Yaskawa INFORM job: FRONT_OST.JBI

/JOB
//NAME FRONT_OST
//POS
///NPOS 25,25,0,5,0,0
///TOOL 0
///POSTYPE PULSE
///PULSE
C00000=27585,-47842,-289,32095,-40789,28095
C00001=4801,-35772,25187,4593,-28023,-82032
C00002=17634,-23800,39238,9573,-31425,-73339
C00003=17634,-23800,39238,9573,-31425,-73339
C00004=16549,-22464,39800,8390,-30730,-72975
C00005=16684,-22641,39722,8536,-30818,-73021
C00006=16684,-19968,45512,8078,-32771,-72767
C00007=17634,-23800,39238,9573,-31425,-73339
C00008=17837,-21535,44509,9322,-33342,-73155
C00009=17837,-21535,44509,9322,-33342,-73155
C00010=16866,-20378,45014,8305,-32755,-72853
C00011=17032,-20588,44918,8481,-32857,-72905
C00012=17032,-17542,51480,8009,-35060,-72636
C00013=17837,-21535,44509,9322,-33342,-73155
C00014=-20829,-18800,50532,-12466,-37179,-77446
C00015=-19934,-17904,50946,-11618,-36715,-77676
C00016=-20044,-18019,50891,-11723,-36773,-77647
C00017=-20044,-15288,56753,-11218,-38713,-77950
C00018=-20966,-18928,50473,-12596,-37250,-77413
C00019=-20884,-26676,33664,-14451,-31668,-76336
C00020=-20884,-26676,33664,-14451,-31668,-76336
C00021=-19557,-25338,34176,-13080,-30873,-76751
C00022=-19691,-25483,34117,-13220,-30955,-76709
C00023=-19691,-22773,39998,-12506,-32911,-77106
C00024=-20642,-26447,33747,-14206,-31526,-76411
BC00000=934475
BC00001=880430
BC00002=895791
BC00003=895791
BC00004=895791
BC00005=895791
BC00006=895791
BC00007=895791
BC00008=900237
BC00009=900237
BC00010=900237
BC00011=900237
BC00012=900237
BC00013=900237
BC00014=900237
BC00015=900237
BC00016=900237
BC00017=900237
BC00018=900237
BC00019=900237
BC00020=900237
BC00021=900237
BC00022=900237
BC00023=900237
BC00024=900237
///POSTYPE BASE
///RECTAN
///RCONF 1,0,0,0,0,0,0,0,0,0,0,0,0,0,0,0,0,0,0,0,0,0,0,0
P00006=0.000,0.000,0.000,0.0000,0.0000,0.0000
///RCONF 0,0,0,0,0,0,0,0,0,0,0,0,0,0,0,0,0,0,0,0,0,0,0,0
P00021=6.550,-0.003,-5.735,0.0000,0.0000,0.0000
P00022=5.943,-0.018,-6.388,0.0000,0.0000,0.0000
P00023=7.025,-0.019,-7.168,0.0000,0.0000,0.0000
P00024=5.926,-0.047,-4.777,0.0000,0.0000,0.0000
//INST
///DATE 2024/05/29 11:52
///ATTR SC,RW
///GROUP1 RB1,BS1
NOP
'POMIAR DO WYJ!! PRZEROBIC NA STD
'KONIEC
MOVJ C00000 BC00000 VJ=25.00
MOVJ C00001 BC00001 VJ=50.00
'W5L
MOVJ C00002 BC00002 VJ=30.00 PL=0
MOVL C00003 BC00003 V=166.7
REFP 3 C00004 BC00004
CALL JOB:SEARCH-R1
SET P0021 P0006
SFTON P0021
MOVL C00005 BC00005 V=166.7
REFP 3 C00006 BC00006
CALL JOB:SEARCH-R1
SET P0021 P0006
SFTON P0021
SFTOF
MOVL C00007 BC00007 V=166.7
'W6L
MOVJ C00008 BC00008 VJ=20.00 PL=0
MOVL C00009 BC00009 V=166.7
REFP 3 C00010 BC00010
CALL JOB:SEARCH-R1
SET P0022 P0006
SFTON P0022
MOVL C00011 BC00011 V=166.7
REFP 3 C00012 BC00012
CALL JOB:SEARCH-R1
SET P0022 P0006
SFTON P0022
SFTOF
MOVL C00013 BC00013 V=166.7
'W6P
MOVL C00014 BC00014 V=333.3 PL=0
REFP 3 C00015 BC00015
CALL JOB:SEARCH-R1
SET P0023 P0006
SFTON P0023
MOVL C00016 BC00016 V=166.7
REFP 3 C00017 BC00017
CALL JOB:SEARCH-R1
SET P0023 P0006
SFTON P0023
SFTOF
MOVL C00018 BC00018 V=166.7
'W5P
MOVJ C00019 BC00019 VJ=20.00 PL=0
MOVL C00020 BC00020 V=166.7
REFP 3 C00021 BC00021
CALL JOB:SEARCH-R1
SET P0024 P0006
SFTON P0024
MOVL C00022 BC00022 V=166.7
REFP 3 C00023 BC00023
CALL JOB:SEARCH-R1
SET P0024 P0006
SFTON P0024
SFTOF
MOVL C00024 BC00024 V=166.7
END
